Staubli VAL3: RosSimpleMsg.pjx

Parameters version=s7.7.2 stackSize=5000 millimeterUnit=true
Program file=start.pgx
Program file=stop.pgx
Data file=RosSimpleMsg.dtx
Type name=Prefix path=../Prefix/Prefix.pjx
Type name=Header path=../Header/Header.pjx
